FUNCTION_BLOCK FB_heightDetection
VAR_INPUT
	
END_VAR
VAR_IN_OUT
	stHeightDetection	: ST_heightDetection;
END_VAR
VAR_OUTPUT
	
END_VAR
VAR
	coeWrt		:	FB_EcCoESdoWrite;
	coeRead		:  	FB_EcCoESdoRead;
	iState	: INT;
	ton_wait : TON;
	heightCmd	: E_HeightDetection;
	height_detection_cmd : E_HeightDetection;//for server to call the method
	iHeight	: DWORD;//0.01mm
END_VAR


coeWrt(
	sNetId:= stHeightDetection.sNetID, 
	nSlaveAddr:=stHeightDetection.nSlaveAddr, 
	nSubIndex:= stHeightDetection.nSubIndex, 
	nIndex:= stHeightDetection.nIndex, 
	pSrcBuf:= ADR(stHeightDetection.iSdoWrite), 
	cbBufLen:= SIZEOF(stHeightDetection.iSdoWrite), 
	bExecute:= , 
	tTimeout:= , 
	bBusy=> , 
	bError=> , 
	nErrId=> );
coeRead(
	sNetId:= stHeightDetection.sNetID, 
	nSlaveAddr:=stHeightDetection.nSlaveAddr, 
	nSubIndex:= stHeightDetection.nSubIndex, 
	nIndex:= stHeightDetection.nIndex, 
	pDstBuf:= ADR(stHeightDetection.iSdoRead), 
	cbBufLen:= SIZEOF(stHeightDetection.iSdoRead), 
	bExecute:= , 
	tTimeout:= , 
	bBusy=> , 
	bError=> , 
	nErrId=> );
ton_wait();
CASE height_detection_cmd OF
	E_HeightDetection.SET_PROGRAM:
		IF M_setProg(iProgram:=16#05) THEN
			height_detection_cmd:= E_HeightDetection.DO_NOTHING;
		END_IF
	E_HeightDetection.READ_HEIGHT:
		IF M_readHeight(iTool:=16#00) THEN
			height_detection_cmd:= E_HeightDetection.DO_NOTHING;
		END_IF	
END_CASE

METHOD M_readHeight : BOOL
VAR_INPUT
	iTool	: DWORD;
END_VAR
VAR_OUTPUT
	
END_VAR
M_readHeight	:= FALSE;
CASE iState OF
	0:
		coeWrt.bExecute	:= FALSE;
		coeRead.bExecute:= FALSE;
		ton_wait.IN	:= FALSE;
		iState	:= 1;
	1://trig
		stHeightDetection.nIndex	:= 16#8005;
		stHeightDetection.nSubIndex	:= 16#01;
		stHeightDetection.iSdoWrite	:= 16#01;
		coeWrt.bExecute	:= TRUE;
		ton_wait.IN	:= TRUE;
		ton_wait.PT:= T#2S;
		IF ton_wait.Q THEN//wait finish
			coeWrt.bExecute	:= FALSE;
			iState	:= 2;
		END_IF			
	2://read tool
		IF NOT coeWrt.bBusy THEN
			stHeightDetection.nIndex	:= 16#8005;
			stHeightDetection.nSubIndex	:= 16#0B;
			stHeightDetection.iSdoWrite	:= iTool;
			coeWrt.bExecute	:= TRUE;
			iState	:= 3;
		END_IF
	3:
		IF coeWrt.bBusy THEN
			coeWrt.bExecute:= FALSE;
			iState	:= 4;
		END_IF
	4://respose of read tool
		IF NOT coeWrt.bBusy THEN
			stHeightDetection.nIndex	:= 16#8005;
			stHeightDetection.nSubIndex	:= 16#0C;		
			coeRead.bExecute	:= TRUE;
			IF coeRead.bBusy THEN
				coeRead.bExecute:= FALSE;
				iState	:= 5;
			END_IF
		END_IF	
	5://read value
		IF NOT coeRead.bBusy THEN
			stHeightDetection.nIndex	:= 16#8005;
			stHeightDetection.nSubIndex	:= 16#0D;		
			coeRead.bExecute	:= TRUE;
			iState	:= 6;
		END_IF
	6:
		IF coeRead.bBusy THEN
			coeRead.bExecute:= FALSE;
			iState	:= 7;
		END_IF
	7:
		IF NOT coeRead.bBusy THEN
			iHeight	:= stHeightDetection.iSdoRead;		
			iState	:= 8;
		END_IF
	8://init trig
		stHeightDetection.nIndex	:= 16#8005;
		stHeightDetection.nSubIndex	:= 16#01;
		stHeightDetection.iSdoWrite	:= 16#00;
		coeWrt.bExecute	:= TRUE;
		IF coeWrt.bBusy THEN
			coeWrt.bExecute	:= FALSE;
			iState	:= 9;
		END_IF
	9:
		IF NOT coeWrt.bBusy THEN
			M_readHeight	:= TRUE;
			iState	:= 0;
		END_IF
				
END_CASE
END_METHOD

METHOD M_setProg : BOOL
VAR_INPUT
	iProgram	: DWORD;
END_VAR
M_setProg	:= FALSE;
CASE iState OF
	0:
		iState	:= 1;
	1:
		stHeightDetection.nIndex	:= 16#8005;
		stHeightDetection.nSubIndex	:= 16#03;
		stHeightDetection.iSdoWrite	:= iProgram;
		coeWrt.bExecute	:= TRUE;
		iState	:= 2;
	2:
		ton_wait.IN := TRUE;
		ton_wait.PT	:= T#1000MS;
		stHeightDetection.nIndex	:= 16#8005;
		stHeightDetection.nSubIndex	:= 16#04;		
		coeRead.bExecute	:= ton_wait.Q;
		IF stHeightDetection.iSdoRead = 1 THEN
			M_setProg	:= TRUE;
			iState	:= 0;
		END_IF
		
		
END_CASE
END_METHOD

END_FUNCTION_BLOCK

(* stored: Version 1.1.0.1, ProductVersion 3.1.4024.12
   POU FB_heightDetection: Id {1279264c-0729-442c-9679-9e1135528f61}, SpecialFunc None
   Method M_readHeight: Id {e432a2ed-0a37-4c1a-ba24-914d5f50cec3}
   Method M_setProg: Id {52bb96c2-4ca7-4a3d-96f2-00e79643c688} *)
